{attribute 'GeneratedUsingTerminal: EL3201-0000-0016'}
{attribute addProperty BoxType "EL3201-0000-0016"}
{attribute addProperty Id "RTD_InputsAT %I*RTD_Inputs_EA9DF21E9WcStateAT %I*WcState_9091E0EB2InfoDataAT %I*InfoData_94A18F5E2"}
{attribute addProperty CRC "3270783690"}
{attribute addProperty Size "13"}
TYPE EL3201_C2F432CA EXTENDS EtcSlaveTerminalBase_947E5A46 :
STRUCT
	{attribute addProperty Name "RTD_Inputs"}
	RTD_Inputs : RTD_Inputs_EA9DF21E;
	{attribute addProperty Name "WcState"}
	WcState : WcState_9091E0EB;
	{attribute addProperty Name "InfoData"}
	InfoData : InfoData_94A18F5E;
END_STRUCT
END_TYPE

(* stored: Version 1.2.0.0, ProductVersion 3.1.4024.9
   DUT EL3201_C2F432CA: Id {68779649-7947-479b-b710-55969a4580d2} *)
